(* IEC 61131-3 sources: TwinCATProj/TwinCATRD/PPS_Archive_fb/Cyl, 23 files *)

(* ---- PPS_Cyl.typ ---- *)
(********************************************************************
 * COPYRIGHT -- Pro Pack Systems, Inc.
 ********************************************************************
 * Library: PPS_Cyl
 * File: PPS_Cyl.typ
 * Author: PaulZ
 * Created: April 16, 2012
 ********************************************************************
 * Data types of library PPS_Cyl
 ********************************************************************)

TYPE
	dtCylCntrlInterface2 : 	STRUCT
		I : dtCylCntrl_Inputs2;
		IQ : dtCylCntrl_InOut2;
		Q : dtCylCntrl_Outputs2;
		stSensorExt : dtDebounceInterface;
		stSensorRet : dtDebounceInterface;
	END_STRUCT;
	dtCylCntrlInterface3 : 	STRUCT
		I : dtCylCntrl_Inputs3;
		IQ : dtCylCntrl_InOut3;
		Q : dtCylCntrl_Outputs3;
		stSensorExt : dtDebounceInterface;
		stSensorRet : dtDebounceInterface;
		stErrData : dtCylCntrl_ErrorData;
	END_STRUCT;
	dtCylCntrl_Inputs2 : 	STRUCT
		xEnableFB : BOOL;
		diType : Enum_CylinderType;
		xValveOffRetract : BOOL;
		xAirOk : BOOL;
		xEnManCntrl : BOOL;
		xManCmdA : BOOL;
		xManCmdB : BOOL;
		xManBrake : BOOL;
		xEmergency : BOOL;
		tTravelDel : TIME;
		xFaultReset : BOOL;
	END_STRUCT;
	dtCylCntrl_Inputs3 : 	STRUCT
		xEnableFB : BOOL;
		diType : Enum_CylinderType;
		xValveOffRetract : BOOL;
		xAirOk : BOOL;
		xEnManCntrl : BOOL;
		xManCmdA : BOOL;
		xManCmdB : BOOL;
		xManBrake : BOOL;
		xEmergency : BOOL;
		tTravelDel : TIME;
		sCylName : STRING[80];
	END_STRUCT;
	dtCylCntrl_InOut2 : 	STRUCT
		xExtCmd : BOOL;
		xRetCmd : BOOL;
		xBrakeEn : BOOL;
		xBrakeDis : BOOL;
	END_STRUCT;
	dtCylCntrl_InOut3 : 	STRUCT
		xExtCmd : BOOL;
		xRetCmd : BOOL;
		xBrakeEn : BOOL;
		xBrakeDis : BOOL;
		xFaultReset : BOOL;
	END_STRUCT;
	dtCylCntrl_Outputs2 : 	STRUCT
		xFBActive : BOOL;
		xSVACmd : BOOL;
		xSVBCmd : BOOL;
		xSVBrakeCmd : BOOL;
		xExtended : BOOL;
		xRetracted : BOOL;
		xFaultNoExt : BOOL;
		xFaultNoRet : BOOL;
		tTimeToExtend : TIME;
		tTimeToRetract : TIME;
	END_STRUCT;
	dtCylCntrl_Outputs3 : 	STRUCT
		xFBActive : BOOL;
		xSVACmd : BOOL;
		xSVBCmd : BOOL;
		xSVBrakeCmd : BOOL;
		xExtended : BOOL;
		xRetracted : BOOL;
		xFault : BOOL;
		sFaultText : STRING[80];
		tTimeToExtend : TIME;
		tTimeToRetract : TIME;
	END_STRUCT;
	dtCylCntrl_ErrorData : 	STRUCT
		uiErrorID : UINT;
	END_STRUCT;
	Enum_CylinderType :
		(
		EN_Cyl_1xSV_Basic := 0,
		EN_Cyl_1xSV_Sensored,
		EN_Cyl_2xSV_Basic_NoBrake,
		EN_Cyl_2xSV_Basic_WBrake,
		EN_Cyl_2xSV_Sensored_NoBrake,
		EN_Cyl_2xSV_Sensored_WBrake
		);
END_TYPE

(* ---- FC_CylFM_1xSV_Basic.st ---- *)
(********************************************************************
 * COPYRIGHT -- Pro Pack Systems, Inc.
 ********************************************************************
 * Library: PPS_Cyl
 * File: FC_CylFM_1xSV_Basic.st
 * Author: PaulZ
 * Created: April 18, 2012
 ********************************************************************
 * Implementation of library PPS_Cyl
 ********************************************************************)

(* Monitors Cylinder Fault for Single SV Cylinder *)
FUNCTION FC_CylFM_1xSV_Basic

IF iq_Cyl.I.diType = EN_Cyl_1xSV_Basic THEN

	IF iq_Cyl.Q.xSVACmd THEN
		IF iq_Timer.Q THEN
			IF iq_Cyl.I.xValveOffRetract THEN
				iq_Cyl.Q.xExtended	:= TRUE;
			ELSE
				iq_Cyl.Q.xRetracted	:= TRUE;
			END_IF
			iq_Timer.IN					:= FALSE;
		END_IF
	ELSE
		IF iq_Timer.Q THEN
			IF iq_Cyl.I.xValveOffRetract THEN
				iq_Cyl.Q.xRetracted	:= TRUE;
			ELSE
				iq_Cyl.Q.xExtended	:= TRUE;
				END_IF
			iq_Timer.IN					:= FALSE;
		END_IF
	END_IF

END_IF

END_FUNCTION

(* ---- FC_CylFM_1xSV_Basic3.st ---- *)
(********************************************************************
 * COPYRIGHT -- Pro Pack Systems, Inc.
 ********************************************************************
 * Library: PPS_Cyl
 * File: FC_CylFM_1xSV_Basic.st
 * Author: PaulZ
 * Created: April 18, 2012
 ********************************************************************
 * Implementation of library PPS_Cyl
 ********************************************************************)

(* Monitors Cylinder Fault for Single SV Cylinder *)
FUNCTION FC_CylFM_1xSV_Basic3

IF iq_Cyl.I.diType = EN_Cyl_1xSV_Basic THEN

	IF iq_Cyl.Q.xSVACmd THEN
		IF iq_Timer.Q THEN
			IF iq_Cyl.I.xValveOffRetract THEN
				iq_Cyl.Q.xExtended	:= TRUE;
			ELSE
				iq_Cyl.Q.xRetracted	:= TRUE;
			END_IF
			iq_Timer.IN					:= FALSE;
		END_IF
	ELSE
		IF iq_Timer.Q THEN
			IF iq_Cyl.I.xValveOffRetract THEN
				iq_Cyl.Q.xRetracted	:= TRUE;
			ELSE
				iq_Cyl.Q.xExtended	:= TRUE;
				END_IF
			iq_Timer.IN					:= FALSE;
		END_IF
	END_IF

END_IF

END_FUNCTION

(* ---- FC_CylFM_1xSV_Sensored.st ---- *)
(********************************************************************
 * COPYRIGHT -- Pro Pack Systems, Inc.
 ********************************************************************
 * Library: PPS_Cyl
 * File: FC_CylFM_1xSV_Sensored.st
 * Author: PaulZ
 * Created: April 18, 2012
 ********************************************************************
 * Implementation of library PPS_Cyl
 ********************************************************************)

(* Monitors Cylinder Fault for Single SV Cylinder with Sensors *)
FUNCTION FC_CylFM_1xSV_Sensored

IF iq_Cyl.I.diType = EN_Cyl_1xSV_Sensored THEN

	xFaultSum	:= iq_Cyl.Q.xFaultNoExt OR iq_Cyl.Q.xFaultNoRet;

	IF NOT xFaultSum THEN
		IF iq_Cyl.I.xValveOffRetract THEN
			IF iq_Cyl.Q.xSVACmd THEN
				IF iq_Cyl.stSensorExt.Q.xCmd THEN
					iq_Cyl.Q.xExtended		:= TRUE;
					iq_Cyl.Q.xFaultNoExt		:= FALSE;
					iq_Timer.IN					:= FALSE;
				ELSE
					IF iq_Timer.Q THEN
						iq_Cyl.Q.xExtended	:= FALSE;
						iq_Cyl.Q.xFaultNoExt	:= TRUE;
						iq_Timer.IN				:= FALSE;
					END_IF
				END_IF
			ELSE
				IF iq_Cyl.stSensorRet.Q.xCmd THEN
					iq_Cyl.Q.xRetracted 		:= TRUE;
					iq_Cyl.Q.xFaultNoRet		:= FALSE;
					iq_Timer.IN					:= FALSE;
				ELSE
					IF iq_Timer.Q THEN
						iq_Cyl.Q.xRetracted	:= FALSE;
						iq_Cyl.Q.xFaultNoRet	:= TRUE;
						iq_Timer.IN				:= FALSE;
					END_IF
				END_IF
			END_IF
		ELSE
			IF NOT iq_Cyl.Q.xSVACmd THEN
				IF iq_Cyl.stSensorExt.Q.xCmd THEN
					iq_Cyl.Q.xExtended		:= TRUE;
					iq_Cyl.Q.xFaultNoExt		:= FALSE;
					iq_Timer.IN					:= FALSE;
				ELSE
					IF iq_Timer.Q THEN
						iq_Cyl.Q.xExtended	:= FALSE;
						iq_Cyl.Q.xFaultNoExt	:= TRUE;
						iq_Timer.IN				:= FALSE;
					END_IF
				END_IF
			ELSE
				IF iq_Cyl.stSensorRet.Q.xCmd THEN
					iq_Cyl.Q.xRetracted		:= TRUE;
					iq_Cyl.Q.xFaultNoRet		:= FALSE;
					iq_Timer.IN					:= FALSE;
				ELSE
					IF iq_Timer.Q THEN
						iq_Cyl.Q.xRetracted	:= FALSE;
						iq_Cyl.Q.xFaultNoRet	:= TRUE;
						iq_Timer.IN				:= FALSE;
					END_IF
				END_IF
			END_IF
		END_IF
	END_IF

END_IF

END_FUNCTION

(* ---- FC_CylFM_1xSV_Sensored3.st ---- *)
(********************************************************************
 * COPYRIGHT -- Pro Pack Systems, Inc.
 ********************************************************************
 * Library: PPS_Cyl
 * File: FC_CylFM_1xSV_Sensored.st
 * Author: PaulZ
 * Created: April 18, 2012
 ********************************************************************
 * Implementation of library PPS_Cyl
 ********************************************************************)

(* Monitors Cylinder Fault for Single SV Cylinder with Sensors *)
FUNCTION FC_CylFM_1xSV_Sensored3

IF iq_Cyl.I.diType = EN_Cyl_1xSV_Sensored THEN

	xFaultSum	:= iq_Cyl.Q.xFault;

	IF NOT xFaultSum THEN
		IF iq_Cyl.I.xValveOffRetract THEN
			IF iq_Cyl.Q.xSVACmd THEN
				IF iq_Cyl.stSensorExt.Q.xCmd THEN
					iq_Cyl.Q.xExtended		:= TRUE;
					iq_Cyl.Q.xFault				:= FALSE;
					iq_Cyl.Q.sFaultText		:= '';
					iq_Timer.IN					:= FALSE;
				ELSE
					IF iq_Timer.Q THEN
						iq_Cyl.Q.xExtended			:= FALSE;
						iq_Cyl.Q.xFault					:= TRUE;
						iq_Cyl.Q.sFaultText			:= CONCAT(iq_Cyl.I.sCylName, sNoExtTxt);
						iq_Timer.IN						:= FALSE;
					END_IF
				END_IF
			ELSE
				IF iq_Cyl.stSensorRet.Q.xCmd THEN
					iq_Cyl.Q.xRetracted 		:= TRUE;
					iq_Cyl.Q.xFault				:= FALSE;
					iq_Cyl.Q.sFaultText		:= '';
					iq_Timer.IN					:= FALSE;
				ELSE
					IF iq_Timer.Q THEN
						iq_Cyl.Q.xRetracted			:= FALSE;
						iq_Cyl.Q.xFault					:= TRUE;
						iq_Cyl.Q.sFaultText			:= CONCAT(iq_Cyl.I.sCylName, sNoRetTxt);
						iq_Timer.IN						:= FALSE;
					END_IF
				END_IF
			END_IF
		ELSE
			IF NOT iq_Cyl.Q.xSVACmd THEN
				IF iq_Cyl.stSensorExt.Q.xCmd THEN
					iq_Cyl.Q.xExtended		:= TRUE;
					iq_Cyl.Q.xFault				:= FALSE;
					iq_Cyl.Q.sFaultText		:= '';
					iq_Timer.IN					:= FALSE;
				ELSE
					IF iq_Timer.Q THEN
						iq_Cyl.Q.xExtended			:= FALSE;
						iq_Cyl.Q.xFault					:= TRUE;
						iq_Cyl.Q.sFaultText			:= CONCAT(iq_Cyl.I.sCylName, sNoExtTxt);
						iq_Timer.IN						:= FALSE;
					END_IF
				END_IF
			ELSE
				IF iq_Cyl.stSensorRet.Q.xCmd THEN
					iq_Cyl.Q.xRetracted		:= TRUE;
					iq_Cyl.Q.xFault				:= FALSE;
					iq_Cyl.Q.sFaultText		:= '';
					iq_Timer.IN					:= FALSE;
				ELSE
					IF iq_Timer.Q THEN
						iq_Cyl.Q.xRetracted			:= FALSE;
						iq_Cyl.Q.xFault					:= TRUE;
						iq_Cyl.Q.sFaultText			:= CONCAT(iq_Cyl.I.sCylName, sNoRetTxt);
						iq_Timer.IN						:= FALSE;
					END_IF
				END_IF
			END_IF
		END_IF
	END_IF

END_IF

END_FUNCTION

(* ---- FC_CylFM_2xSV_Basic_NoBrake.st ---- *)
(********************************************************************
 * COPYRIGHT -- Pro Pack Systems, Inc.
 ********************************************************************
 * Library: PPS_Cyl
 * File: FC_CylFM_2xSV_Basic_NoBrake.st
 * Author: PaulZ
 * Created: April 18, 2012
 ********************************************************************
 * Implementation of library PPS_Cyl
 ********************************************************************)

(* Monitors Cylinder Fault for Double SV Cylinder *)
FUNCTION FC_CylFM_2xSV_Basic_NoBrake

IF iq_Cyl.I.diType = EN_Cyl_2xSV_Basic_NoBrake THEN

	IF iq_Cyl.Q.xSVACmd THEN
		IF iq_Timer.Q THEN
			IF iq_Cyl.I.xValveOffRetract THEN
				iq_Cyl.Q.xExtended		:= TRUE;
				iq_Cyl.Q.tTimeToExtend	:= iq_Timer.ET;
			ELSE
				iq_Cyl.Q.xRetracted		:= TRUE;
				iq_Cyl.Q.tTimeToRetract	:= iq_Timer.ET;
			END_IF
			iq_Timer.IN						:= FALSE;
		END_IF
	ELSIF iq_Cyl.Q.xSVBCmd THEN
		IF iq_Timer.Q THEN
			IF iq_Cyl.I.xValveOffRetract THEN
				iq_Cyl.Q.xRetracted		:= TRUE;
				iq_Cyl.Q.tTimeToRetract	:= iq_Timer.ET;
			ELSE
				iq_Cyl.Q.xExtended		:= TRUE;
				iq_Cyl.Q.tTimeToExtend	:= iq_Timer.ET;
 			END_IF
			iq_Timer.IN						:= FALSE;
		END_IF
	END_IF

END_IF

END_FUNCTION

(* ---- FC_CylFM_2xSV_Basic_NoBrake3.st ---- *)
(********************************************************************
 * COPYRIGHT -- Pro Pack Systems, Inc.
 ********************************************************************
 * Library: PPS_Cyl
 * File: FC_CylFM_2xSV_Basic_NoBrake.st
 * Author: PaulZ
 * Created: April 18, 2012
 ********************************************************************
 * Implementation of library PPS_Cyl
 ********************************************************************)

(* Monitors Cylinder Fault for Double SV Cylinder *)
FUNCTION FC_CylFM_2xSV_Basic_NoBrake3

IF iq_Cyl.I.diType = EN_Cyl_2xSV_Basic_NoBrake THEN

	IF iq_Cyl.Q.xSVACmd THEN
		IF iq_Timer.Q THEN
			IF iq_Cyl.I.xValveOffRetract THEN
				iq_Cyl.Q.xExtended		:= TRUE;
				iq_Cyl.Q.tTimeToExtend	:= iq_Timer.ET;
			ELSE
				iq_Cyl.Q.xRetracted		:= TRUE;
				iq_Cyl.Q.tTimeToRetract	:= iq_Timer.ET;
			END_IF
			iq_Timer.IN						:= FALSE;
		END_IF
	ELSIF iq_Cyl.Q.xSVBCmd THEN
		IF iq_Timer.Q THEN
			IF iq_Cyl.I.xValveOffRetract THEN
				iq_Cyl.Q.xRetracted		:= TRUE;
				iq_Cyl.Q.tTimeToRetract	:= iq_Timer.ET;
			ELSE
				iq_Cyl.Q.xExtended		:= TRUE;
				iq_Cyl.Q.tTimeToExtend	:= iq_Timer.ET;
 			END_IF
			iq_Timer.IN						:= FALSE;
		END_IF
	END_IF

END_IF

END_FUNCTION

(* ---- FC_CylFM_2xSV_Basic_wBrake.st ---- *)
(********************************************************************
 * COPYRIGHT -- Pro Pack Systems, Inc.
 ********************************************************************
 * Library: PPS_Cyl
 * File: FC_CylFM_2xSV_Basic_wBrake.st
 * Author: PaulZ
 * Created: April 23, 2012
 ********************************************************************
 * Implementation of library PPS_Cyl
 ********************************************************************)

(* Monitors Cylinder Faults for Double SV Cylinder, no Sensors, with Brake *)
FUNCTION FC_CylFM_2xSV_Basic_wBrake

IF iq_Cyl.I.diType = EN_Cyl_2xSV_Basic_WBrake THEN

	IF iq_Cyl.Q.xSVACmd THEN
		IF iq_Timer.Q THEN
			IF iq_Cyl.I.xValveOffRetract THEN
				iq_Cyl.Q.xExtended		:= TRUE;
				iq_Cyl.Q.tTimeToExtend	:= iq_Timer.ET;
			ELSE
				iq_Cyl.Q.xRetracted		:= TRUE;
				iq_Cyl.Q.tTimeToRetract	:= iq_Timer.ET;
			END_IF
			iq_Timer.IN						:= FALSE;
		END_IF
	ELSIF iq_Cyl.Q.xSVBCmd THEN
		IF iq_Timer.Q THEN
			IF iq_Cyl.I.xValveOffRetract THEN
				iq_Cyl.Q.xRetracted		:= TRUE;
				iq_Cyl.Q.tTimeToRetract	:= iq_Timer.ET;
			ELSE
				iq_Cyl.Q.xExtended		:= TRUE;
				iq_Cyl.Q.tTimeToExtend	:= iq_Timer.ET;
 			END_IF
			iq_Timer.IN						:= FALSE;
		END_IF
	END_IF

END_IF

END_FUNCTION

(* ---- FC_CylFM_2xSV_Basic_wBrake3.st ---- *)
(********************************************************************
 * COPYRIGHT -- Pro Pack Systems, Inc.
 ********************************************************************
 * Library: PPS_Cyl
 * File: FC_CylFM_2xSV_Basic_wBrake.st
 * Author: PaulZ
 * Created: April 23, 2012
 ********************************************************************
 * Implementation of library PPS_Cyl
 ********************************************************************)

(* Monitors Cylinder Faults for Double SV Cylinder, no Sensors, with Brake *)
FUNCTION FC_CylFM_2xSV_Basic_wBrake3

IF iq_Cyl.I.diType = EN_Cyl_2xSV_Basic_WBrake THEN

	IF iq_Cyl.Q.xSVACmd THEN
		IF iq_Timer.Q THEN
			IF iq_Cyl.I.xValveOffRetract THEN
				iq_Cyl.Q.xExtended		:= TRUE;
				iq_Cyl.Q.tTimeToExtend	:= iq_Timer.ET;
			ELSE
				iq_Cyl.Q.xRetracted		:= TRUE;
				iq_Cyl.Q.tTimeToRetract	:= iq_Timer.ET;
			END_IF
			iq_Timer.IN						:= FALSE;
		END_IF
	ELSIF iq_Cyl.Q.xSVBCmd THEN
		IF iq_Timer.Q THEN
			IF iq_Cyl.I.xValveOffRetract THEN
				iq_Cyl.Q.xRetracted		:= TRUE;
				iq_Cyl.Q.tTimeToRetract	:= iq_Timer.ET;
			ELSE
				iq_Cyl.Q.xExtended		:= TRUE;
				iq_Cyl.Q.tTimeToExtend	:= iq_Timer.ET;
 			END_IF
			iq_Timer.IN						:= FALSE;
		END_IF
	END_IF

END_IF

END_FUNCTION

(* ---- FC_CylFM_2xSV_Sensored_NoBrake.st ---- *)
(********************************************************************
 * COPYRIGHT -- Pro Pack Systems, Inc.
 ********************************************************************
 * Library: PPS_Cyl
 * File: FC_CylFM_2xSV_Sensored_NoBrake.st
 * Author: PaulZ
 * Created: April 18, 2012
 ********************************************************************
 * Implementation of library PPS_Cyl
 ********************************************************************)

(* Monitors Cylinder Fault for Double SV Cylinder with Sensor and no Brake *)
FUNCTION FC_CylFM_2xSV_Sensored_NoBrake

IF iq_Cyl.I.diType = EN_Cyl_2xSV_Sensored_NoBrake THEN

	xFaultSum	:= iq_Cyl.Q.xFaultNoExt OR iq_Cyl.Q.xFaultNoRet;

 	IF NOT xFaultSum THEN
		IF iq_Cyl.I.xValveOffRetract THEN
			IF iq_Cyl.Q.xSVACmd THEN
				IF iq_Cyl.stSensorExt.Q.xCmd THEN
					iq_Cyl.Q.xExtended			:= TRUE;
					iq_Cyl.Q.xFaultNoExt			:= FALSE;
					iq_Timer.IN						:= FALSE;
				ELSE
					IF iq_Timer.Q THEN
						iq_Cyl.Q.xExtended		:= FALSE;
						iq_Cyl.Q.xFaultNoExt		:= TRUE;
						iq_Timer.IN					:= FALSE;
					END_IF
				END_IF
			ELSIF iq_Cyl.Q.xSVBCmd THEN
				IF iq_Cyl.stSensorRet.Q.xCmd THEN
					iq_Cyl.Q.xRetracted 			:= TRUE;
					iq_Cyl.Q.xFaultNoRet			:= FALSE;
					iq_Timer.IN						:= FALSE;
				ELSE
					IF iq_Timer.Q THEN
						iq_Cyl.Q.xRetracted		:= FALSE;
						iq_Cyl.Q.xFaultNoRet		:= TRUE;
						iq_Timer.IN					:= FALSE;
					END_IF
				END_IF
			END_IF
		ELSE
			IF iq_Cyl.Q.xSVBCmd THEN
				IF iq_Cyl.stSensorExt.Q.xCmd THEN
					iq_Cyl.Q.xExtended			:= TRUE;
					iq_Cyl.Q.xFaultNoExt			:= FALSE;
					iq_Timer.IN						:= FALSE;
				ELSE
					IF iq_Timer.Q THEN
						iq_Cyl.Q.xExtended		:= FALSE;
						iq_Cyl.Q.xFaultNoExt		:= TRUE;
						iq_Timer.IN					:= FALSE;
					END_IF
				END_IF
			ELSIF iq_Cyl.Q.xSVACmd THEN
				IF iq_Cyl.stSensorRet.Q.xCmd THEN
					iq_Cyl.Q.xRetracted			:= TRUE;
					iq_Cyl.Q.xFaultNoRet			:= FALSE;
					iq_Timer.IN						:= FALSE;
				ELSE
					IF iq_Timer.Q THEN
						iq_Cyl.Q.xRetracted		:= FALSE;
						iq_Cyl.Q.xFaultNoRet		:= TRUE;
						iq_Timer.IN					:= FALSE;
					END_IF
				END_IF
			END_IF
		END_IF
	END_IF

END_IF

END_FUNCTION

(* ---- FC_CylFM_2xSV_Sensored_NoBrake3.st ---- *)
(********************************************************************
 * COPYRIGHT -- Pro Pack Systems, Inc.
 ********************************************************************
 * Library: PPS_Cyl
 * File: FC_CylFM_2xSV_Sensored_NoBrake.st
 * Author: PaulZ
 * Created: April 18, 2012
 ********************************************************************
 * Implementation of library PPS_Cyl
 ********************************************************************)

(* Monitors Cylinder Fault for Double SV Cylinder with Sensor and no Brake *)
FUNCTION FC_CylFM_2xSV_Sensored_NoBrake3

IF iq_Cyl.I.diType = EN_Cyl_2xSV_Sensored_NoBrake THEN

	xFaultSum	:= iq_Cyl.Q.xFault;

 	IF NOT xFaultSum THEN
		IF iq_Cyl.I.xValveOffRetract THEN
			IF iq_Cyl.Q.xSVACmd THEN
				IF iq_Cyl.stSensorExt.Q.xCmd THEN
					iq_Cyl.Q.xExtended			:= TRUE;
					iq_Cyl.Q.xFault					:= FALSE;
					iq_Cyl.Q.sFaultText			:= '';
					iq_Timer.IN						:= FALSE;
				ELSE
					IF iq_Timer.Q THEN
						iq_Cyl.Q.xExtended			:= FALSE;
						iq_Cyl.Q.xFault					:= TRUE;
						iq_Cyl.Q.sFaultText			:= CONCAT(iq_Cyl.I.sCylName, sNoExtTxt);
						iq_Timer.IN						:= FALSE;
					END_IF
				END_IF
			ELSIF iq_Cyl.Q.xSVBCmd THEN
				IF iq_Cyl.stSensorRet.Q.xCmd THEN
					iq_Cyl.Q.xRetracted 			:= TRUE;
					iq_Cyl.Q.xFault					:= FALSE;
					iq_Cyl.Q.sFaultText			:= '';
					iq_Timer.IN						:= FALSE;
				ELSE
					IF iq_Timer.Q THEN
						iq_Cyl.Q.xRetracted			:= FALSE;
						iq_Cyl.Q.xFault					:= TRUE;
						iq_Cyl.Q.sFaultText			:= CONCAT(iq_Cyl.I.sCylName, sNoRetTxt);
						iq_Timer.IN						:= FALSE;
					END_IF
				END_IF
			END_IF
		ELSE
			IF iq_Cyl.Q.xSVBCmd THEN
				IF iq_Cyl.stSensorExt.Q.xCmd THEN
					iq_Cyl.Q.xExtended			:= TRUE;
					iq_Cyl.Q.xFault					:= FALSE;
					iq_Cyl.Q.sFaultText			:= '';
					iq_Timer.IN						:= FALSE;
				ELSE
					IF iq_Timer.Q THEN
						iq_Cyl.Q.xExtended			:= FALSE;
						iq_Cyl.Q.xFault					:= TRUE;
						iq_Cyl.Q.sFaultText			:= CONCAT(iq_Cyl.I.sCylName, sNoExtTxt);
						iq_Timer.IN						:= FALSE;
					END_IF
				END_IF
			ELSIF iq_Cyl.Q.xSVACmd THEN
				IF iq_Cyl.stSensorRet.Q.xCmd THEN
					iq_Cyl.Q.xRetracted			:= TRUE;
					iq_Cyl.Q.xFault					:= FALSE;
					iq_Cyl.Q.sFaultText			:= '';
					iq_Timer.IN						:= FALSE;
				ELSE
					IF iq_Timer.Q THEN
						iq_Cyl.Q.xRetracted			:= FALSE;
						iq_Cyl.Q.xFault					:= TRUE;
						iq_Cyl.Q.sFaultText			:= CONCAT(iq_Cyl.I.sCylName, sNoRetTxt);
						iq_Timer.IN						:= FALSE;
					END_IF
				END_IF
			END_IF
		END_IF
	END_IF

END_IF

END_FUNCTION

(* ---- FC_CylFM_2xSV_Sensored_wBrake.st ---- *)
(********************************************************************
 * COPYRIGHT -- Pro Pack Systems, Inc.
 ********************************************************************
 * Library: PPS_Cyl
 * File: FC_CylFM_2xSV_Sensored_wBrake.st
 * Author: PaulZ
 * Created: April 18, 2012
 ********************************************************************
 * Implementation of library PPS_Cyl
 ********************************************************************)

(* Monitors Cylinder Fault for Double SV Cylinder with Sensors and Brake *)
FUNCTION FC_CylFM_2xSV_Sensored_wBrake

IF iq_Cyl.I.diType = EN_Cyl_2xSV_Sensored_WBrake THEN

	xFaultSum	:= iq_Cyl.Q.xFaultNoExt OR iq_Cyl.Q.xFaultNoRet;

 	IF iq_Cyl.Q.xSVBrakeCmd THEN
 		iq_Timer.IN		:= FALSE;
	END_IF

	IF NOT xFaultSum THEN
		IF iq_Cyl.I.xValveOffRetract THEN
			IF iq_Cyl.Q.xSVACmd THEN
				IF iq_Cyl.stSensorExt.Q.xCmd THEN
					iq_Cyl.Q.xExtended			:= TRUE;
					iq_Cyl.Q.xFaultNoExt			:= FALSE;
					iq_Timer.IN						:= FALSE;
				ELSE
					IF iq_Timer.Q THEN
						iq_Cyl.Q.xExtended		:= FALSE;
						iq_Cyl.Q.xFaultNoExt		:= TRUE;
						iq_Timer.IN					:= FALSE;
					END_IF
				END_IF
			ELSIF iq_Cyl.Q.xSVBCmd THEN
				IF iq_Cyl.stSensorRet.Q.xCmd THEN
					iq_Cyl.Q.xRetracted 			:= TRUE;
					iq_Cyl.Q.xFaultNoRet			:= FALSE;
					iq_Timer.IN						:= FALSE;
				ELSE
					IF iq_Timer.Q THEN
						iq_Cyl.Q.xRetracted		:= FALSE;
						iq_Cyl.Q.xFaultNoRet		:= TRUE;
						iq_Timer.IN					:= FALSE;
					END_IF
				END_IF
			END_IF
		ELSE
			IF iq_Cyl.Q.xSVBCmd THEN
				IF iq_Cyl.stSensorExt.Q.xCmd THEN
					iq_Cyl.Q.xExtended			:= TRUE;
					iq_Cyl.Q.xFaultNoExt			:= FALSE;
					iq_Timer.IN						:= FALSE;
				ELSE
					IF iq_Timer.Q THEN
						iq_Cyl.Q.xExtended		:= FALSE;
						iq_Cyl.Q.xFaultNoExt		:= TRUE;
						iq_Timer.IN					:= FALSE;
					END_IF
				END_IF
			ELSIF iq_Cyl.Q.xSVACmd THEN
				IF iq_Cyl.stSensorRet.Q.xCmd THEN
					iq_Cyl.Q.xRetracted			:= TRUE;
					iq_Cyl.Q.xFaultNoRet			:= FALSE;
					iq_Timer.IN						:= FALSE;
				ELSE
					IF iq_Timer.Q THEN
						iq_Cyl.Q.xRetracted		:= FALSE;
						iq_Cyl.Q.xFaultNoRet		:= TRUE;
						iq_Timer.IN					:= FALSE;
					END_IF
				END_IF
			END_IF
		END_IF
	END_IF

END_IF

END_FUNCTION

(* ---- FC_CylFM_2xSV_Sensored_wBrake3.st ---- *)
(********************************************************************
 * COPYRIGHT -- Pro Pack Systems, Inc.
 ********************************************************************
 * Library: PPS_Cyl
 * File: FC_CylFM_2xSV_Sensored_wBrake.st
 * Author: PaulZ
 * Created: April 18, 2012
 ********************************************************************
 * Implementation of library PPS_Cyl
 ********************************************************************)

(* Monitors Cylinder Fault for Double SV Cylinder with Sensors and Brake *)
FUNCTION FC_CylFM_2xSV_Sensored_wBrake3

IF iq_Cyl.I.diType = EN_Cyl_2xSV_Sensored_WBrake THEN

	xFaultSum	:= iq_Cyl.Q.xFault;

 	IF iq_Cyl.Q.xSVBrakeCmd THEN
 		iq_Timer.IN		:= FALSE;
	END_IF

	IF NOT xFaultSum THEN
		IF iq_Cyl.I.xValveOffRetract THEN
			IF iq_Cyl.Q.xSVACmd THEN
				IF iq_Cyl.stSensorExt.Q.xCmd THEN
					iq_Cyl.Q.xExtended			:= TRUE;
					iq_Cyl.Q.xFault					:= FALSE;
					iq_Cyl.Q.sFaultText			:= '';
					iq_Timer.IN						:= FALSE;
				ELSE
					IF iq_Timer.Q THEN
						iq_Cyl.Q.xExtended			:= FALSE;
						iq_Cyl.Q.xFault					:= TRUE;
						iq_Cyl.Q.sFaultText			:= CONCAT(iq_Cyl.I.sCylName, sNoExtTxt);
						iq_Timer.IN						:= FALSE;
					END_IF
				END_IF
			ELSIF iq_Cyl.Q.xSVBCmd THEN
				IF iq_Cyl.stSensorRet.Q.xCmd THEN
					iq_Cyl.Q.xRetracted 			:= TRUE;
					iq_Cyl.Q.xFault					:= FALSE;
					iq_Cyl.Q.sFaultText			:= '';
					iq_Timer.IN						:= FALSE;
				ELSE
					IF iq_Timer.Q THEN
						iq_Cyl.Q.xRetracted			:= FALSE;
						iq_Cyl.Q.xFault					:= TRUE;
						iq_Cyl.Q.sFaultText			:= CONCAT(iq_Cyl.I.sCylName, sNoRetTxt);
						iq_Timer.IN						:= FALSE;
					END_IF
				END_IF
			END_IF
		ELSE
			IF iq_Cyl.Q.xSVBCmd THEN
				IF iq_Cyl.stSensorExt.Q.xCmd THEN
					iq_Cyl.Q.xExtended			:= TRUE;
					iq_Cyl.Q.xFault					:= FALSE;
					iq_Cyl.Q.sFaultText			:= '';
					iq_Timer.IN						:= FALSE;
				ELSE
					IF iq_Timer.Q THEN
						iq_Cyl.Q.xExtended			:= FALSE;
						iq_Cyl.Q.xFault					:= TRUE;
						iq_Cyl.Q.sFaultText			:= CONCAT(iq_Cyl.I.sCylName, sNoExtTxt);
						iq_Timer.IN						:= FALSE;
					END_IF
				END_IF
			ELSIF iq_Cyl.Q.xSVACmd THEN
				IF iq_Cyl.stSensorRet.Q.xCmd THEN
					iq_Cyl.Q.xRetracted			:= TRUE;
					iq_Cyl.Q.xFault					:= FALSE;
					iq_Cyl.Q.sFaultText			:= '';
					iq_Timer.IN						:= FALSE;
				ELSE
					IF iq_Timer.Q THEN
						iq_Cyl.Q.xRetracted			:= FALSE;
						iq_Cyl.Q.xFault					:= TRUE;
						iq_Cyl.Q.sFaultText			:= CONCAT(iq_Cyl.I.sCylName, sNoRetTxt);
						iq_Timer.IN						:= FALSE;
					END_IF
				END_IF
			END_IF
		END_IF
	END_IF

END_IF

END_FUNCTION

(* ---- FC_CylQ_1xSV.st ---- *)
(********************************************************************
 * COPYRIGHT -- Pro Pack Systems, Inc.
 ********************************************************************
 * Library: PPS_Cyl
 * File: FC_CylQ_1xSV_Basic.st
 * Author: PaulZ
 * Created: April 19, 2012
 ********************************************************************
 * Implementation of library PPS_Cyl
 ********************************************************************)

(* Controls the outputs for a Single SV Cylinder *)
FUNCTION FC_CylQ_1xSV

IF iq_Cyl.I.diType = EN_Cyl_1xSV_Basic OR
	iq_Cyl.I.diType = EN_Cyl_1xSV_Sensored THEN

	IF NOT iq_Cyl.I.xEnManCntrl THEN (* When not in Manual Mode, control output *)

		IF iq_Cyl.I.xValveOffRetract THEN
			IF iq_Cyl.IQ.xExtCmd THEN
				iq_Cyl.Q.xSVACmd		:= TRUE;
				iq_Cyl.Q.xRetracted		:= FALSE;
				iq_Cyl.Q.xExtended		:= FALSE;
				iq_Cyl.Q.tTimeToExtend	:= T#0ms;
				iq_Timer.IN					:= TRUE;
				IF iq_Cyl.Q.xSVACmd THEN
					iq_Cyl.IQ.xExtCmd		:= FALSE;
				END_IF
			END_IF

			IF iq_Cyl.IQ.xRetCmd THEN
				iq_Cyl.Q.xSVACmd		:= FALSE;
				iq_Cyl.Q.xExtended		:= FALSE;
				iq_Cyl.Q.xRetracted		:= FALSE;
				iq_Cyl.Q.tTimeToRetract	:= T#0ms;
				iq_Timer.IN					:= TRUE;
				IF NOT iq_Cyl.Q.xSVACmd THEN
					iq_Cyl.IQ.xRetCmd		:= FALSE;
				END_IF
			END_IF
		ELSE
			IF iq_Cyl.IQ.xExtCmd THEN
				iq_Cyl.Q.xSVACmd		:= FALSE;
				iq_Cyl.Q.xExtended		:= FALSE;
				iq_Cyl.Q.xRetracted		:= FALSE;
				iq_Cyl.Q.tTimeToExtend	:= T#0ms;
				iq_Timer.IN					:= TRUE;
				IF NOT iq_Cyl.Q.xSVACmd THEN
					iq_Cyl.IQ.xExtCmd		:= FALSE;
				END_IF
			END_IF

			IF iq_Cyl.IQ.xRetCmd THEN
				iq_Cyl.Q.xSVACmd		:= TRUE;
				iq_Cyl.Q.xExtended		:= FALSE;
				iq_Cyl.Q.xRetracted		:= FALSE;
				iq_Cyl.Q.tTimeToRetract	:= T#0ms;
				iq_Timer.IN					:= TRUE;
				IF iq_Cyl.Q.xSVACmd THEN
					iq_Cyl.IQ.xRetCmd		:= FALSE;
				END_IF
			END_IF
		END_IF

	ELSE (* When in Manual Mode, control output *)
		IF iq_Cyl.Q.xSVACmd THEN
			IF xManCmd THEN
				iq_Cyl.Q.xSVACmd		:= FALSE;
				iq_Cyl.Q.xRetracted		:= FALSE;
				iq_Cyl.Q.xExtended		:= FALSE;
				iq_Cyl.Q.tTimeToRetract	:= T#0ms;
				iq_Timer.IN					:= TRUE;
			END_IF
		ELSE
			IF xManCmd THEN
				iq_Cyl.Q.xSVACmd		:= TRUE;
				iq_Cyl.Q.xRetracted		:= FALSE;
				iq_Cyl.Q.xExtended		:= FALSE;
				iq_Cyl.Q.tTimeToExtend	:= T#0ms;
				iq_Timer.IN					:= TRUE;
			END_IF
		END_IF
	END_IF

END_IF

END_FUNCTION

(* ---- FC_CylQ_1xSV3.st ---- *)
(********************************************************************
 * COPYRIGHT -- Pro Pack Systems, Inc.
 ********************************************************************
 * Library: PPS_Cyl
 * File: FC_CylQ_1xSV_Basic.st
 * Author: PaulZ
 * Created: April 19, 2012
 ********************************************************************
 * Implementation of library PPS_Cyl
 ********************************************************************)

(* Controls the outputs for a Single SV Cylinder *)
FUNCTION FC_CylQ_1xSV3

IF iq_Cyl.I.diType = EN_Cyl_1xSV_Basic OR
	iq_Cyl.I.diType = EN_Cyl_1xSV_Sensored THEN

	IF NOT iq_Cyl.I.xEnManCntrl THEN (* When not in Manual Mode, control output *)

		IF iq_Cyl.I.xValveOffRetract THEN
			IF iq_Cyl.IQ.xExtCmd THEN
				iq_Cyl.Q.xSVACmd		:= TRUE;
				iq_Cyl.Q.xRetracted		:= FALSE;
				iq_Cyl.Q.xExtended		:= FALSE;
				iq_Cyl.Q.tTimeToExtend	:= T#0ms;
				iq_Timer.IN					:= TRUE;
				IF iq_Cyl.Q.xSVACmd THEN
					iq_Cyl.IQ.xExtCmd		:= FALSE;
				END_IF
			END_IF

			IF iq_Cyl.IQ.xRetCmd THEN
				iq_Cyl.Q.xSVACmd		:= FALSE;
				iq_Cyl.Q.xExtended		:= FALSE;
				iq_Cyl.Q.xRetracted		:= FALSE;
				iq_Cyl.Q.tTimeToRetract	:= T#0ms;
				iq_Timer.IN					:= TRUE;
				IF NOT iq_Cyl.Q.xSVACmd THEN
					iq_Cyl.IQ.xRetCmd		:= FALSE;
				END_IF
			END_IF
		ELSE
			IF iq_Cyl.IQ.xExtCmd THEN
				iq_Cyl.Q.xSVACmd		:= FALSE;
				iq_Cyl.Q.xExtended		:= FALSE;
				iq_Cyl.Q.xRetracted		:= FALSE;
				iq_Cyl.Q.tTimeToExtend	:= T#0ms;
				iq_Timer.IN					:= TRUE;
				IF NOT iq_Cyl.Q.xSVACmd THEN
					iq_Cyl.IQ.xExtCmd		:= FALSE;
				END_IF
			END_IF

			IF iq_Cyl.IQ.xRetCmd THEN
				iq_Cyl.Q.xSVACmd		:= TRUE;
				iq_Cyl.Q.xExtended		:= FALSE;
				iq_Cyl.Q.xRetracted		:= FALSE;
				iq_Cyl.Q.tTimeToRetract	:= T#0ms;
				iq_Timer.IN					:= TRUE;
				IF iq_Cyl.Q.xSVACmd THEN
					iq_Cyl.IQ.xRetCmd		:= FALSE;
				END_IF
			END_IF
		END_IF

	ELSE (* When in Manual Mode, control output *)
		IF iq_Cyl.Q.xSVACmd THEN
			IF xManCmd THEN
				iq_Cyl.Q.xSVACmd		:= FALSE;
				iq_Cyl.Q.xRetracted		:= FALSE;
				iq_Cyl.Q.xExtended		:= FALSE;
				iq_Cyl.Q.tTimeToRetract	:= T#0ms;
				iq_Timer.IN					:= TRUE;
			END_IF
		ELSE
			IF xManCmd THEN
				iq_Cyl.Q.xSVACmd		:= TRUE;
				iq_Cyl.Q.xRetracted		:= FALSE;
				iq_Cyl.Q.xExtended		:= FALSE;
				iq_Cyl.Q.tTimeToExtend	:= T#0ms;
				iq_Timer.IN					:= TRUE;
			END_IF
		END_IF
	END_IF

END_IF

END_FUNCTION

(* ---- FC_CylQ_2xSV_NoBrake.st ---- *)
(********************************************************************
 * COPYRIGHT -- Pro Pack Systems, Inc.
 ********************************************************************
 * Library: PPS_Cyl
 * File: FC_CylQ_1xSV_Basic.st
 * Author: PaulZ
 * Created: April 19, 2012
 ********************************************************************
 * Implementation of library PPS_Cyl
 ********************************************************************)

(* Controls the outputs for a Double SV Cylinder, no Brake *)
FUNCTION FC_CylQ_2xSV_NoBrake

IF iq_Cyl.I.diType = EN_Cyl_2xSV_Basic_NoBrake OR
	iq_Cyl.I.diType = EN_Cyl_2xSV_Sensored_NoBrake THEN

	IF NOT iq_Cyl.I.xEnManCntrl THEN (* When not in Manual Mode, control output *)

		IF iq_Cyl.I.xValveOffRetract THEN
			IF iq_Cyl.IQ.xExtCmd THEN
				iq_Cyl.Q.xSVACmd		:= TRUE;
				iq_Cyl.Q.xSVBCmd		:= FALSE;
				iq_Cyl.Q.xRetracted		:= FALSE;
				iq_Cyl.Q.xExtended		:= FALSE;
				iq_Cyl.Q.tTimeToExtend	:= T#0ms;
				iq_Timer.IN					:= TRUE;
				IF iq_Cyl.Q.xSVACmd AND NOT iq_Cyl.Q.xSVBCmd THEN
					iq_Cyl.IQ.xExtCmd		:= FALSE;
				END_IF
			END_IF

			IF iq_Cyl.IQ.xRetCmd THEN
				iq_Cyl.Q.xSVACmd		:= FALSE;
				iq_Cyl.Q.xSVBCmd		:= TRUE;
				iq_Cyl.Q.xExtended		:= FALSE;
				iq_Cyl.Q.xRetracted		:= FALSE;
				iq_Cyl.Q.tTimeToRetract	:= T#0ms;
				iq_Timer.IN					:= TRUE;
				IF NOT iq_Cyl.Q.xSVACmd AND iq_Cyl.Q.xSVBCmd THEN
					iq_Cyl.IQ.xRetCmd		:= FALSE;
				END_IF
			END_IF
		ELSE
			IF iq_Cyl.IQ.xExtCmd THEN
				iq_Cyl.Q.xSVACmd		:= FALSE;
				iq_Cyl.Q.xSVBCmd		:= TRUE;
				iq_Cyl.Q.xExtended		:= FALSE;
				iq_Cyl.Q.xRetracted		:= FALSE;
				iq_Cyl.Q.tTimeToExtend	:= T#0ms;
				iq_Timer.IN					:= TRUE;
				IF NOT iq_Cyl.Q.xSVACmd AND iq_Cyl.Q.xSVBCmd THEN
					iq_Cyl.IQ.xExtCmd		:= FALSE;
				END_IF
			END_IF

			IF iq_Cyl.IQ.xRetCmd THEN
				iq_Cyl.Q.xSVACmd		:= TRUE;
				iq_Cyl.Q.xSVBCmd		:= FALSE;
				iq_Cyl.Q.xExtended		:= FALSE;
				iq_Cyl.Q.xRetracted		:= FALSE;
				iq_Cyl.Q.tTimeToRetract	:= T#0ms;
				iq_Timer.IN					:= TRUE;
				IF iq_Cyl.Q.xSVACmd AND NOT iq_Cyl.Q.xSVBCmd THEN
					iq_Cyl.IQ.xRetCmd		:= FALSE;
				END_IF
			END_IF
		END_IF

	ELSE (* When in Manual Mode, control output *)
		IF iq_Cyl.Q.xSVACmd THEN
			IF xManCmd THEN
				iq_Cyl.Q.xSVACmd		:= FALSE;
				iq_Cyl.Q.xRetracted		:= FALSE;
				iq_Cyl.Q.xExtended		:= FALSE;
				iq_Timer.IN					:= TRUE;
			END_IF
		ELSE
			IF xManCmd THEN
				iq_Cyl.Q.xSVACmd		:= TRUE;
				iq_Cyl.Q.xSVBCmd		:= FALSE;
				iq_Cyl.Q.xRetracted		:= FALSE;
				iq_Cyl.Q.xExtended		:= FALSE;
				IF iq_Cyl.I.xValveOffRetract THEN
					iq_Cyl.Q.tTimeToExtend	:= T#0ms;
				ELSE
					iq_Cyl.Q.tTimeToRetract	:= T#0ms;
	 			END_IF
				iq_Timer.IN					:= TRUE;
			END_IF
		END_IF

		IF iq_Cyl.Q.xSVBCmd THEN
			IF xManCmdB THEN
				iq_Cyl.Q.xSVBCmd		:= FALSE;
				iq_Cyl.Q.xRetracted		:= FALSE;
				iq_Cyl.Q.xExtended		:= FALSE;
				iq_Timer.IN					:= TRUE;
			END_IF
		ELSE
			IF xManCmdB THEN
				iq_Cyl.Q.xSVBCmd		:= TRUE;
				iq_Cyl.Q.xSVACmd		:= FALSE;
				iq_Cyl.Q.xRetracted		:= FALSE;
				iq_Cyl.Q.xExtended		:= FALSE;
				IF iq_Cyl.I.xValveOffRetract THEN
					iq_Cyl.Q.tTimeToRetract	:= T#0ms;
				ELSE
					iq_Cyl.Q.tTimeToExtend	:= T#0ms;
	 			END_IF
				iq_Timer.IN					:= TRUE;
			END_IF
		END_IF
	END_IF

END_IF

END_FUNCTION

(* ---- FC_CylQ_2xSV_NoBrake3.st ---- *)
(********************************************************************
 * COPYRIGHT -- Pro Pack Systems, Inc.
 ********************************************************************
 * Library: PPS_Cyl
 * File: FC_CylQ_1xSV_Basic.st
 * Author: PaulZ
 * Created: April 19, 2012
 ********************************************************************
 * Implementation of library PPS_Cyl
 ********************************************************************)

(* Controls the outputs for a Double SV Cylinder, no Brake *)
FUNCTION FC_CylQ_2xSV_NoBrake3

IF iq_Cyl.I.diType = EN_Cyl_2xSV_Basic_NoBrake OR
	iq_Cyl.I.diType = EN_Cyl_2xSV_Sensored_NoBrake THEN

	IF NOT iq_Cyl.I.xEnManCntrl THEN (* When not in Manual Mode, control output *)

		IF iq_Cyl.I.xValveOffRetract THEN
			IF iq_Cyl.IQ.xExtCmd THEN
				iq_Cyl.Q.xSVACmd		:= TRUE;
				iq_Cyl.Q.xSVBCmd		:= FALSE;
				iq_Cyl.Q.xRetracted		:= FALSE;
				iq_Cyl.Q.xExtended		:= FALSE;
				iq_Cyl.Q.tTimeToExtend	:= T#0ms;
				iq_Timer.IN					:= TRUE;
				IF iq_Cyl.Q.xSVACmd AND NOT iq_Cyl.Q.xSVBCmd THEN
					iq_Cyl.IQ.xExtCmd		:= FALSE;
				END_IF
			END_IF

			IF iq_Cyl.IQ.xRetCmd THEN
				iq_Cyl.Q.xSVACmd		:= FALSE;
				iq_Cyl.Q.xSVBCmd		:= TRUE;
				iq_Cyl.Q.xExtended		:= FALSE;
				iq_Cyl.Q.xRetracted		:= FALSE;
				iq_Cyl.Q.tTimeToRetract	:= T#0ms;
				iq_Timer.IN					:= TRUE;
				IF NOT iq_Cyl.Q.xSVACmd AND iq_Cyl.Q.xSVBCmd THEN
					iq_Cyl.IQ.xRetCmd		:= FALSE;
				END_IF
			END_IF
		ELSE
			IF iq_Cyl.IQ.xExtCmd THEN
				iq_Cyl.Q.xSVACmd		:= FALSE;
				iq_Cyl.Q.xSVBCmd		:= TRUE;
				iq_Cyl.Q.xExtended		:= FALSE;
				iq_Cyl.Q.xRetracted		:= FALSE;
				iq_Cyl.Q.tTimeToExtend	:= T#0ms;
				iq_Timer.IN					:= TRUE;
				IF NOT iq_Cyl.Q.xSVACmd AND iq_Cyl.Q.xSVBCmd THEN
					iq_Cyl.IQ.xExtCmd		:= FALSE;
				END_IF
			END_IF

			IF iq_Cyl.IQ.xRetCmd THEN
				iq_Cyl.Q.xSVACmd		:= TRUE;
				iq_Cyl.Q.xSVBCmd		:= FALSE;
				iq_Cyl.Q.xExtended		:= FALSE;
				iq_Cyl.Q.xRetracted		:= FALSE;
				iq_Cyl.Q.tTimeToRetract	:= T#0ms;
				iq_Timer.IN					:= TRUE;
				IF iq_Cyl.Q.xSVACmd AND NOT iq_Cyl.Q.xSVBCmd THEN
					iq_Cyl.IQ.xRetCmd		:= FALSE;
				END_IF
			END_IF
		END_IF

	ELSE (* When in Manual Mode, control output *)
		IF iq_Cyl.Q.xSVACmd THEN
			IF xManCmd THEN
				iq_Cyl.Q.xSVACmd		:= FALSE;
				iq_Cyl.Q.xRetracted		:= FALSE;
				iq_Cyl.Q.xExtended		:= FALSE;
				iq_Timer.IN					:= TRUE;
			END_IF
		ELSE
			IF xManCmd THEN
				iq_Cyl.Q.xSVACmd		:= TRUE;
				iq_Cyl.Q.xSVBCmd		:= FALSE;
				iq_Cyl.Q.xRetracted		:= FALSE;
				iq_Cyl.Q.xExtended		:= FALSE;
				IF iq_Cyl.I.xValveOffRetract THEN
					iq_Cyl.Q.tTimeToExtend	:= T#0ms;
				ELSE
					iq_Cyl.Q.tTimeToRetract	:= T#0ms;
	 			END_IF
				iq_Timer.IN					:= TRUE;
			END_IF
		END_IF

		IF iq_Cyl.Q.xSVBCmd THEN
			IF xManCmdB THEN
				iq_Cyl.Q.xSVBCmd		:= FALSE;
				iq_Cyl.Q.xRetracted		:= FALSE;
				iq_Cyl.Q.xExtended		:= FALSE;
				iq_Timer.IN					:= TRUE;
			END_IF
		ELSE
			IF xManCmdB THEN
				iq_Cyl.Q.xSVBCmd		:= TRUE;
				iq_Cyl.Q.xSVACmd		:= FALSE;
				iq_Cyl.Q.xRetracted		:= FALSE;
				iq_Cyl.Q.xExtended		:= FALSE;
				IF iq_Cyl.I.xValveOffRetract THEN
					iq_Cyl.Q.tTimeToRetract	:= T#0ms;
				ELSE
					iq_Cyl.Q.tTimeToExtend	:= T#0ms;
	 			END_IF
				iq_Timer.IN					:= TRUE;
			END_IF
		END_IF
	END_IF

END_IF

END_FUNCTION

(* ---- FC_CylQ_2xSV_wBrake.st ---- *)
(********************************************************************
 * COPYRIGHT -- Pro Pack Systems, Inc.
 ********************************************************************
 * Library: PPS_Cyl
 * File: FC_CylQ_1xSV_Basic.st
 * Author: PaulZ
 * Created: April 19, 2012
 ********************************************************************
 * Implementation of library PPS_Cyl
 ********************************************************************)

(* Controls the outputs for a Double SV Cylinder, with Brake *)
FUNCTION FC_CylQ_2xSV_wBrake

IF iq_Cyl.I.diType = EN_Cyl_2xSV_Basic_WBrake OR
	iq_Cyl.I.diType = EN_Cyl_2xSV_Sensored_WBrake THEN

	IF NOT iq_Cyl.I.xEnManCntrl THEN (* When not in Manual Mode, control output *)

		IF iq_Cyl.IQ.xBrakeEn THEN
  			iq_Cyl.Q.xSVACmd		:= FALSE;
   			iq_Cyl.Q.xSVBCmd		:= FALSE;
   			iq_Cyl.Q.xSVBrakeCmd	:= TRUE;
			iq_Timer.IN					:= FALSE;
			iq_Cyl.IQ.xBrakeEn		:= FALSE;
   		END_IF

		IF iq_Cyl.IQ.xBrakeDis THEN
  			iq_Cyl.Q.xSVBrakeCmd	:= FALSE;
   			iq_Cyl.IQ.xBrakeDis		:= FALSE;
   		END_IF

		IF iq_Cyl.Q.xSVBrakeCmd THEN
  			iq_Cyl.IQ.xExtCmd		:= FALSE;
   			iq_Cyl.IQ.xRetCmd		:= FALSE;
   		END_IF

		IF iq_Cyl.I.xValveOffRetract THEN
			IF iq_Cyl.IQ.xExtCmd THEN
				iq_Cyl.Q.xSVACmd		:= TRUE;
				iq_Cyl.Q.xSVBCmd		:= FALSE;
				iq_Cyl.Q.xRetracted		:= FALSE;
				iq_Cyl.Q.xExtended		:= FALSE;
				iq_Cyl.Q.tTimeToExtend	:= T#0ms;
				iq_Timer.IN					:= TRUE;
				IF iq_Cyl.Q.xSVACmd AND NOT iq_Cyl.Q.xSVBCmd THEN
					iq_Cyl.IQ.xExtCmd		:= FALSE;
				END_IF
			END_IF

			IF iq_Cyl.IQ.xRetCmd THEN
				iq_Cyl.Q.xSVACmd		:= FALSE;
				iq_Cyl.Q.xSVBCmd		:= TRUE;
				iq_Cyl.Q.xExtended		:= FALSE;
				iq_Cyl.Q.xRetracted		:= FALSE;
				iq_Cyl.Q.tTimeToRetract	:= T#0ms;
				iq_Timer.IN					:= TRUE;
				IF NOT iq_Cyl.Q.xSVACmd AND iq_Cyl.Q.xSVBCmd THEN
					iq_Cyl.IQ.xRetCmd		:= FALSE;
				END_IF
			END_IF
		ELSE
			IF iq_Cyl.IQ.xExtCmd THEN
				iq_Cyl.Q.xSVACmd		:= FALSE;
				iq_Cyl.Q.xSVBCmd		:= TRUE;
				iq_Cyl.Q.xExtended		:= FALSE;
				iq_Cyl.Q.xRetracted		:= FALSE;
				iq_Cyl.Q.tTimeToExtend	:= T#0ms;
				iq_Timer.IN					:= TRUE;
				IF NOT iq_Cyl.Q.xSVACmd AND iq_Cyl.Q.xSVBCmd THEN
					iq_Cyl.IQ.xExtCmd		:= FALSE;
				END_IF
			END_IF

			IF iq_Cyl.IQ.xRetCmd THEN
				iq_Cyl.Q.xSVACmd		:= TRUE;
				iq_Cyl.Q.xSVBCmd		:= FALSE;
				iq_Cyl.Q.xExtended		:= FALSE;
				iq_Cyl.Q.xRetracted		:= FALSE;
				iq_Cyl.Q.tTimeToRetract	:= T#0ms;
				iq_Timer.IN					:= TRUE;
				IF iq_Cyl.Q.xSVACmd AND NOT iq_Cyl.Q.xSVBCmd THEN
					iq_Cyl.IQ.xRetCmd		:= FALSE;
				END_IF
			END_IF
		END_IF

	ELSE (* When in Manual Mode, control output *)

		IF xManBrake THEN
  			IF iq_Cyl.Q.xSVBrakeCmd THEN
   				iq_Cyl.Q.xSVBrakeCmd	:= FALSE;
			ELSE
			  	iq_Cyl.Q.xSVBrakeCmd	:= TRUE;
				iq_Cyl.Q.xSVACmd		:= FALSE;
				iq_Cyl.Q.xSVBCmd		:= FALSE;
			END_IF
		END_IF

		IF iq_Cyl.Q.xSVACmd THEN
			IF xManCmd THEN
				iq_Cyl.Q.xSVACmd		:= FALSE;
				iq_Cyl.Q.xRetracted		:= FALSE;
				iq_Cyl.Q.xExtended		:= FALSE;
				iq_Timer.IN					:= TRUE;
			END_IF
		ELSE
			IF xManCmd THEN
				iq_Cyl.Q.xSVACmd		:= TRUE;
				iq_Cyl.Q.xSVBCmd		:= FALSE;
				iq_Cyl.Q.xRetracted		:= FALSE;
				iq_Cyl.Q.xExtended		:= FALSE;
				IF iq_Cyl.I.xValveOffRetract THEN
					iq_Cyl.Q.tTimeToExtend	:= T#0ms;
	 			ELSE
					iq_Cyl.Q.tTimeToRetract	:= T#0ms;
	 			END_IF
				iq_Timer.IN					:= TRUE;
			END_IF
		END_IF

		IF iq_Cyl.Q.xSVBCmd THEN
			IF xManCmdB THEN
				iq_Cyl.Q.xSVBCmd		:= FALSE;
				iq_Cyl.Q.xRetracted		:= FALSE;
				iq_Cyl.Q.xExtended		:= FALSE;
				iq_Timer.IN					:= TRUE;
			END_IF
		ELSE
			IF xManCmdB THEN
				iq_Cyl.Q.xSVBCmd		:= TRUE;
				iq_Cyl.Q.xSVACmd		:= FALSE;
				iq_Cyl.Q.xRetracted		:= FALSE;
				iq_Cyl.Q.xExtended		:= FALSE;
				IF iq_Cyl.I.xValveOffRetract THEN
					iq_Cyl.Q.tTimeToRetract	:= T#0ms;
	 			ELSE
					iq_Cyl.Q.tTimeToExtend	:= T#0ms;
	 			END_IF
				iq_Timer.IN					:= TRUE;
			END_IF
		END_IF
	END_IF

END_IF

END_FUNCTION

(* ---- FC_CylQ_2xSV_wBrake3.st ---- *)
(********************************************************************
 * COPYRIGHT -- Pro Pack Systems, Inc.
 ********************************************************************
 * Library: PPS_Cyl
 * File: FC_CylQ_1xSV_Basic.st
 * Author: PaulZ
 * Created: April 19, 2012
 ********************************************************************
 * Implementation of library PPS_Cyl
 ********************************************************************)

(* Controls the outputs for a Double SV Cylinder, with Brake *)
FUNCTION FC_CylQ_2xSV_wBrake3

IF iq_Cyl.I.diType = EN_Cyl_2xSV_Basic_WBrake OR
	iq_Cyl.I.diType = EN_Cyl_2xSV_Sensored_WBrake THEN

	IF NOT iq_Cyl.I.xEnManCntrl THEN (* When not in Manual Mode, control output *)

		IF iq_Cyl.IQ.xBrakeEn THEN
  			iq_Cyl.Q.xSVACmd		:= FALSE;
   			iq_Cyl.Q.xSVBCmd		:= FALSE;
   			iq_Cyl.Q.xSVBrakeCmd	:= TRUE;
			iq_Timer.IN					:= FALSE;
			iq_Cyl.IQ.xBrakeEn		:= FALSE;
   		END_IF

		IF iq_Cyl.IQ.xBrakeDis THEN
  			iq_Cyl.Q.xSVBrakeCmd	:= FALSE;
   			iq_Cyl.IQ.xBrakeDis		:= FALSE;
   		END_IF

		IF iq_Cyl.Q.xSVBrakeCmd THEN
  			iq_Cyl.IQ.xExtCmd		:= FALSE;
   			iq_Cyl.IQ.xRetCmd		:= FALSE;
   		END_IF

		IF iq_Cyl.I.xValveOffRetract THEN
			IF iq_Cyl.IQ.xExtCmd THEN
				iq_Cyl.Q.xSVACmd		:= TRUE;
				iq_Cyl.Q.xSVBCmd		:= FALSE;
				iq_Cyl.Q.xRetracted		:= FALSE;
				iq_Cyl.Q.xExtended		:= FALSE;
				iq_Cyl.Q.tTimeToExtend	:= T#0ms;
				iq_Timer.IN					:= TRUE;
				IF iq_Cyl.Q.xSVACmd AND NOT iq_Cyl.Q.xSVBCmd THEN
					iq_Cyl.IQ.xExtCmd		:= FALSE;
				END_IF
			END_IF

			IF iq_Cyl.IQ.xRetCmd THEN
				iq_Cyl.Q.xSVACmd		:= FALSE;
				iq_Cyl.Q.xSVBCmd		:= TRUE;
				iq_Cyl.Q.xExtended		:= FALSE;
				iq_Cyl.Q.xRetracted		:= FALSE;
				iq_Cyl.Q.tTimeToRetract	:= T#0ms;
				iq_Timer.IN					:= TRUE;
				IF NOT iq_Cyl.Q.xSVACmd AND iq_Cyl.Q.xSVBCmd THEN
					iq_Cyl.IQ.xRetCmd		:= FALSE;
				END_IF
			END_IF
		ELSE
			IF iq_Cyl.IQ.xExtCmd THEN
				iq_Cyl.Q.xSVACmd		:= FALSE;
				iq_Cyl.Q.xSVBCmd		:= TRUE;
				iq_Cyl.Q.xExtended		:= FALSE;
				iq_Cyl.Q.xRetracted		:= FALSE;
				iq_Cyl.Q.tTimeToExtend	:= T#0ms;
				iq_Timer.IN					:= TRUE;
				IF NOT iq_Cyl.Q.xSVACmd AND iq_Cyl.Q.xSVBCmd THEN
					iq_Cyl.IQ.xExtCmd		:= FALSE;
				END_IF
			END_IF

			IF iq_Cyl.IQ.xRetCmd THEN
				iq_Cyl.Q.xSVACmd		:= TRUE;
				iq_Cyl.Q.xSVBCmd		:= FALSE;
				iq_Cyl.Q.xExtended		:= FALSE;
				iq_Cyl.Q.xRetracted		:= FALSE;
				iq_Cyl.Q.tTimeToRetract	:= T#0ms;
				iq_Timer.IN					:= TRUE;
				IF iq_Cyl.Q.xSVACmd AND NOT iq_Cyl.Q.xSVBCmd THEN
					iq_Cyl.IQ.xRetCmd		:= FALSE;
				END_IF
			END_IF
		END_IF

	ELSE (* When in Manual Mode, control output *)

		IF xManBrake THEN
  			IF iq_Cyl.Q.xSVBrakeCmd THEN
   				iq_Cyl.Q.xSVBrakeCmd	:= FALSE;
			ELSE
			  	iq_Cyl.Q.xSVBrakeCmd	:= TRUE;
				iq_Cyl.Q.xSVACmd		:= FALSE;
				iq_Cyl.Q.xSVBCmd		:= FALSE;
			END_IF
		END_IF

		IF iq_Cyl.Q.xSVACmd THEN
			IF xManCmd THEN
				iq_Cyl.Q.xSVACmd		:= FALSE;
				iq_Cyl.Q.xRetracted		:= FALSE;
				iq_Cyl.Q.xExtended		:= FALSE;
				iq_Timer.IN					:= TRUE;
			END_IF
		ELSE
			IF xManCmd THEN
				iq_Cyl.Q.xSVACmd		:= TRUE;
				iq_Cyl.Q.xSVBCmd		:= FALSE;
				iq_Cyl.Q.xRetracted		:= FALSE;
				iq_Cyl.Q.xExtended		:= FALSE;
				IF iq_Cyl.I.xValveOffRetract THEN
					iq_Cyl.Q.tTimeToExtend	:= T#0ms;
	 			ELSE
					iq_Cyl.Q.tTimeToRetract	:= T#0ms;
	 			END_IF
				iq_Timer.IN					:= TRUE;
			END_IF
		END_IF

		IF iq_Cyl.Q.xSVBCmd THEN
			IF xManCmdB THEN
				iq_Cyl.Q.xSVBCmd		:= FALSE;
				iq_Cyl.Q.xRetracted		:= FALSE;
				iq_Cyl.Q.xExtended		:= FALSE;
				iq_Timer.IN					:= TRUE;
			END_IF
		ELSE
			IF xManCmdB THEN
				iq_Cyl.Q.xSVBCmd		:= TRUE;
				iq_Cyl.Q.xSVACmd		:= FALSE;
				iq_Cyl.Q.xRetracted		:= FALSE;
				iq_Cyl.Q.xExtended		:= FALSE;
				IF iq_Cyl.I.xValveOffRetract THEN
					iq_Cyl.Q.tTimeToRetract	:= T#0ms;
	 			ELSE
					iq_Cyl.Q.tTimeToExtend	:= T#0ms;
	 			END_IF
				iq_Timer.IN					:= TRUE;
			END_IF
		END_IF
	END_IF

END_IF

END_FUNCTION

(* ---- FB_CylCntrl2.st ---- *)
(********************************************************************
 * COPYRIGHT -- Pro Pack Systems, Inc.
 ********************************************************************
 * Library: PPS_Cyl
 * File: FB_CylCntrl2.st
 * Author: Paul Zurlinden
 * Created: April 16, 2012
 ********************************************************************
 * Implementation of library PPS_Cyl
 ********************************************************************)

(* Controls a pneumatic cylinder of the following types:
		EN_Cyl_1xSV_Basic
		EN_Cyl_1xSV_Sensored
		EN_Cyl_2xSV_Basic_NoBrake
		EN_Cyl_2xSV_Basic_WBrake
		EN_Cyl_2xSV_Sensored_NoBrake
		EN_Cyl_2xSV_Sensored_WBrake *)

FUNCTION_BLOCK FB_CylCntrl2

xMonitor :=	iq_CylCntrlInterface.I.diType = EN_Cyl_1xSV_Sensored OR
					iq_CylCntrlInterface.I.diType = EN_Cyl_2xSV_Sensored_NoBrake OR
					iq_CylCntrlInterface.I.diType = EN_Cyl_2xSV_Sensored_WBrake;

x2xSV	:= iq_CylCntrlInterface.I.diType = EN_Cyl_2xSV_Basic_NoBrake OR
				iq_CylCntrlInterface.I.diType = EN_Cyl_2xSV_Basic_WBrake OR
				iq_CylCntrlInterface.I.diType = EN_Cyl_2xSV_Sensored_NoBrake OR
				iq_CylCntrlInterface.I.diType = EN_Cyl_2xSV_Sensored_WBrake;

Timer(PT := iq_CylCntrlInterface.I.tTravelDel);

RT(CLK := iq_CylCntrlInterface.I.xManCmdA);
xManCmd	:= RT.Q;

RT_B(CLK := iq_CylCntrlInterface.I.xManCmdB);
xManCmdB := RT_B.Q;

RT_Brake(CLK := iq_CylCntrlInterface.I.xManBrake);
xManBrake := RT_Brake.Q;

RT_Air(CLK := iq_CylCntrlInterface.I.xAirOk);
FT_Air(CLK := iq_CylCntrlInterface.I.xAirOk);

(* Debounce Cylinder Position Sensors *)
IF xMonitor THEN
	aFB_SensExt[0](iq_DebounceInterface := iq_CylCntrlInterface.stSensorExt);
	aFB_SensExt[1](iq_DebounceInterface := iq_CylCntrlInterface.stSensorRet);

	RT_SensExt(CLK := iq_CylCntrlInterface.stSensorExt.I.xSignal);
	IF RT_SensExt.Q THEN
 		iq_CylCntrlInterface.Q.tTimeToExtend	:= Timer.ET;
	END_IF

	RT_SensRet(CLK := iq_CylCntrlInterface.stSensorRet.I.xSignal);
	IF RT_SensRet.Q THEN
 		iq_CylCntrlInterface.Q.tTimeToRetract	:= Timer.ET;
	END_IF
END_IF

xFaultSum	:= iq_CylCntrlInterface.Q.xFaultNoExt OR iq_CylCntrlInterface.Q.xFaultNoRet;

IF iq_CylCntrlInterface.I.xFaultReset THEN
	iq_CylCntrlInterface.Q.xFaultNoExt	:= FALSE;
	iq_CylCntrlInterface.Q.xFaultNoRet := FALSE;
END_IF

IF iq_CylCntrlInterface.I.xEnableFB THEN
	iq_CylCntrlInterface.Q.xFBActive	:= TRUE;

	(* Determine Cylinder Position when air is first turned on *)
	CASE iCheckAir OF
 		0:
			IF RT_Air.Q THEN
   				IF xMonitor OR x2xSV THEN
   					iCheckAir	:= 10;
				ELSE
					IF iq_CylCntrlInterface.I.xValveOffRetract THEN
   						IF iq_CylCntrlInterface.Q.xSVACmd THEN
							iq_CylCntrlInterface.Q.xExtended	:= TRUE;
							iq_CylCntrlInterface.Q.xRetracted	:= FALSE;
	 					ELSE
						   	iq_CylCntrlInterface.Q.xRetracted	:= TRUE;
							iq_CylCntrlInterface.Q.xExtended	:= FALSE;
	 					END_IF
					ELSE
						IF iq_CylCntrlInterface.Q.xSVACmd THEN
							iq_CylCntrlInterface.Q.xRetracted	:= TRUE;
							iq_CylCntrlInterface.Q.xExtended	:= FALSE;
	 					ELSE
						   	iq_CylCntrlInterface.Q.xExtended	:= TRUE;
							iq_CylCntrlInterface.Q.xRetracted	:= FALSE;
		 				END_IF
					END_IF
				END_IF
			END_IF

		10:
			IF xMonitor THEN
   				iCheckAir	:= 20;
			ELSE
				IF iq_CylCntrlInterface.I.xValveOffRetract THEN
   					IF iq_CylCntrlInterface.Q.xSVACmd THEN
						iq_CylCntrlInterface.Q.xExtended	:= TRUE;
						iq_CylCntrlInterface.Q.xRetracted	:= FALSE;
						iCheckAir										:= 0;
	 				ELSIF iq_CylCntrlInterface.Q.xSVBCmd THEN
					   	iq_CylCntrlInterface.Q.xRetracted	:= TRUE;
						iq_CylCntrlInterface.Q.xExtended	:= FALSE;
						iCheckAir										:= 0;
	 				END_IF
				ELSE
					IF iq_CylCntrlInterface.Q.xSVACmd THEN
						iq_CylCntrlInterface.Q.xRetracted	:= TRUE;
						iq_CylCntrlInterface.Q.xExtended	:= FALSE;
						iCheckAir										:= 0;
	 				ELSIF iq_CylCntrlInterface.Q.xSVBCmd THEN
					   	iq_CylCntrlInterface.Q.xExtended	:= TRUE;
						iq_CylCntrlInterface.Q.xRetracted	:= FALSE;
						iCheckAir										:= 0;
		 			END_IF
				END_IF
			END_IF

		20:
			IF iq_CylCntrlInterface.stSensorExt.Q.xCmd THEN
   				iq_CylCntrlInterface.Q.xExtended	:= TRUE;
				iq_CylCntrlInterface.Q.xRetracted	:= FALSE;
				iCheckAir										:= 0;
			END_IF

			IF iq_CylCntrlInterface.stSensorRet.Q.xCmd THEN
   				iq_CylCntrlInterface.Q.xRetracted	:= TRUE;
				iq_CylCntrlInterface.Q.xExtended	:= FALSE;
				iCheckAir										:= 0;
			END_IF

	END_CASE

	(* Fault Montiors *)
	FC_CylFM_1xSV_Basic(iq_CylCntrlInterface, Timer);
	FC_CylFM_1xSV_Sensored(iq_CylCntrlInterface, Timer);
	FC_CylFM_2xSV_Basic_NoBrake(iq_CylCntrlInterface, Timer);
	FC_CylFM_2xSV_Basic_wBrake(iq_CylCntrlInterface, Timer);
	FC_CylFM_2xSV_Sensored_NoBrake(iq_CylCntrlInterface, Timer);
	FC_CylFM_2xSV_Sensored_wBrake(iq_CylCntrlInterface, Timer);

	(* Control output *)
	IF iq_CylCntrlInterface.I.xEmergency OR xFaultSum OR FT_Air.Q THEN
		iq_CylCntrlInterface.Q.xSVACmd			:= FALSE;
		iq_CylCntrlInterface.Q.xSVBCmd			:= FALSE;
		iq_CylCntrlInterface.Q.xSVBrakeCmd	:= FALSE;
	ELSE
		FC_CylQ_1xSV(xManCmd, iq_CylCntrlInterface, Timer);
		FC_CylQ_2xSV_NoBrake(xManCmd, xManCmdB, iq_CylCntrlInterface, Timer);
		FC_CylQ_2xSV_wBrake(xManCmd, xManCmdB, xManBrake, iq_CylCntrlInterface, Timer);
	END_IF

	IF iq_CylCntrlInterface.I.xEmergency THEN
 		iq_CylCntrlInterface.Q.xExtended	:= FALSE;
  		iq_CylCntrlInterface.Q.xRetracted	:= FALSE;
  	END_IF

ELSE
	iq_CylCntrlInterface.Q.xFBActive			:= FALSE;
	iq_CylCntrlInterface.Q.xSVACmd			:= FALSE;
	iq_CylCntrlInterface.Q.xSVBCmd			:= FALSE;
 	iq_CylCntrlInterface.Q.xSVBrakeCmd	:= FALSE;
	iq_CylCntrlInterface.Q.xExtended		:= FALSE;
	iq_CylCntrlInterface.Q.xRetracted		:= FALSE;
	Timer.IN											:= FALSE;
END_IF

END_FUNCTION_BLOCK

(* ---- FB_CylCntrl3.st ---- *)
(********************************************************************
 * COPYRIGHT -- Pro Pack Systems, Inc.
 ********************************************************************
 * Library: PPS_Cyl
 * File: FB_CylCntrl3.st
 * Author: PaulZ
 * Created: March 14, 2013
 ********************************************************************
 * Implementation of library PPS_Cyl
 ********************************************************************)

(* Controls a pneumatic cylinder of the following types:
		EN_Cyl_1xSV_Basic
		EN_Cyl_1xSV_Sensored
		EN_Cyl_2xSV_Basic_NoBrake
		EN_Cyl_2xSV_Basic_WBrake
		EN_Cyl_2xSV_Sensored_NoBrake
		EN_Cyl_2xSV_Sensored_WBrake *)

FUNCTION_BLOCK FB_CylCntrl3

xMonitor :=	iq_CylCntrlInterface.I.diType = EN_Cyl_1xSV_Sensored OR
					iq_CylCntrlInterface.I.diType = EN_Cyl_2xSV_Sensored_NoBrake OR
					iq_CylCntrlInterface.I.diType = EN_Cyl_2xSV_Sensored_WBrake;

x2xSV	:= iq_CylCntrlInterface.I.diType = EN_Cyl_2xSV_Basic_NoBrake OR
				iq_CylCntrlInterface.I.diType = EN_Cyl_2xSV_Basic_WBrake OR
				iq_CylCntrlInterface.I.diType = EN_Cyl_2xSV_Sensored_NoBrake OR
				iq_CylCntrlInterface.I.diType = EN_Cyl_2xSV_Sensored_WBrake;

Timer(PT := iq_CylCntrlInterface.I.tTravelDel);

RT(CLK := iq_CylCntrlInterface.I.xManCmdA);
xManCmd	:= RT.Q;

RT_B(CLK := iq_CylCntrlInterface.I.xManCmdB);
xManCmdB := RT_B.Q;

RT_Brake(CLK := iq_CylCntrlInterface.I.xManBrake);
xManBrake := RT_Brake.Q;

RT_Air(CLK := iq_CylCntrlInterface.I.xAirOk);
FT_Air(CLK := iq_CylCntrlInterface.I.xAirOk);

(* Debounce Cylinder Position Sensors *)
IF xMonitor THEN
	aFB_SensExt[0](iq_DebounceInterface := iq_CylCntrlInterface.stSensorExt);
	aFB_SensExt[1](iq_DebounceInterface := iq_CylCntrlInterface.stSensorRet);

	RT_SensExt(CLK := iq_CylCntrlInterface.stSensorExt.I.xSignal);
	IF RT_SensExt.Q THEN
 		iq_CylCntrlInterface.Q.tTimeToExtend	:= Timer.ET;
	END_IF

	RT_SensRet(CLK := iq_CylCntrlInterface.stSensorRet.I.xSignal);
	IF RT_SensRet.Q THEN
 		iq_CylCntrlInterface.Q.tTimeToRetract	:= Timer.ET;
	END_IF
END_IF

xFaultSum	:= iq_CylCntrlInterface.Q.xFault;

IF iq_CylCntrlInterface.IQ.xFaultReset THEN
	iq_CylCntrlInterface.Q.xFault			:= FALSE;
	iq_CylCntrlInterface.Q.sFaultText		:= '';
	iq_CylCntrlInterface.IQ.xFaultReset		:= FALSE;
END_IF

IF iq_CylCntrlInterface.I.xEnableFB THEN
	iq_CylCntrlInterface.Q.xFBActive	:= TRUE;

	(* Determine Cylinder Position when air is first turned on *)
	CASE iCheckAir OF
 		0:
			IF RT_Air.Q THEN
   				IF xMonitor OR x2xSV THEN
   					iCheckAir	:= 10;
				ELSE
					IF iq_CylCntrlInterface.I.xValveOffRetract THEN
   						IF iq_CylCntrlInterface.Q.xSVACmd THEN
							iq_CylCntrlInterface.Q.xExtended	:= TRUE;
							iq_CylCntrlInterface.Q.xRetracted	:= FALSE;
	 					ELSE
						   	iq_CylCntrlInterface.Q.xRetracted	:= TRUE;
							iq_CylCntrlInterface.Q.xExtended	:= FALSE;
	 					END_IF
					ELSE
						IF iq_CylCntrlInterface.Q.xSVACmd THEN
							iq_CylCntrlInterface.Q.xRetracted	:= TRUE;
							iq_CylCntrlInterface.Q.xExtended	:= FALSE;
	 					ELSE
						   	iq_CylCntrlInterface.Q.xExtended	:= TRUE;
							iq_CylCntrlInterface.Q.xRetracted	:= FALSE;
		 				END_IF
					END_IF
				END_IF
			END_IF

		10:
			IF xMonitor THEN
   				iCheckAir	:= 20;
			ELSE
				IF iq_CylCntrlInterface.I.xValveOffRetract THEN
   					IF iq_CylCntrlInterface.Q.xSVACmd THEN
						iq_CylCntrlInterface.Q.xExtended	:= TRUE;
						iq_CylCntrlInterface.Q.xRetracted	:= FALSE;
						iCheckAir										:= 0;
	 				ELSIF iq_CylCntrlInterface.Q.xSVBCmd THEN
					   	iq_CylCntrlInterface.Q.xRetracted	:= TRUE;
						iq_CylCntrlInterface.Q.xExtended	:= FALSE;
						iCheckAir										:= 0;
	 				END_IF
				ELSE
					IF iq_CylCntrlInterface.Q.xSVACmd THEN
						iq_CylCntrlInterface.Q.xRetracted	:= TRUE;
						iq_CylCntrlInterface.Q.xExtended	:= FALSE;
						iCheckAir										:= 0;
	 				ELSIF iq_CylCntrlInterface.Q.xSVBCmd THEN
					   	iq_CylCntrlInterface.Q.xExtended	:= TRUE;
						iq_CylCntrlInterface.Q.xRetracted	:= FALSE;
						iCheckAir										:= 0;
		 			END_IF
				END_IF
			END_IF

		20:
			IF iq_CylCntrlInterface.stSensorExt.Q.xCmd THEN
   				iq_CylCntrlInterface.Q.xExtended	:= TRUE;
				iq_CylCntrlInterface.Q.xRetracted	:= FALSE;
				iCheckAir										:= 0;
			END_IF

			IF iq_CylCntrlInterface.stSensorRet.Q.xCmd THEN
   				iq_CylCntrlInterface.Q.xRetracted	:= TRUE;
				iq_CylCntrlInterface.Q.xExtended	:= FALSE;
				iCheckAir										:= 0;
			END_IF

	END_CASE

	(* Fault Montiors *)
	FC_CylFM_1xSV_Basic3(iq_CylCntrlInterface, Timer);
	FC_CylFM_1xSV_Sensored3(iq_CylCntrlInterface, Timer);
	FC_CylFM_2xSV_Basic_NoBrake3(iq_CylCntrlInterface, Timer);
	FC_CylFM_2xSV_Basic_wBrake3(iq_CylCntrlInterface, Timer);
	FC_CylFM_2xSV_Sensored_NoBrake3(iq_CylCntrlInterface, Timer);
	FC_CylFM_2xSV_Sensored_wBrake3(iq_CylCntrlInterface, Timer);

	(* Control output *)
	IF iq_CylCntrlInterface.I.xEmergency OR xFaultSum OR FT_Air.Q THEN
		iq_CylCntrlInterface.Q.xSVACmd			:= FALSE;
		iq_CylCntrlInterface.Q.xSVBCmd			:= FALSE;
		iq_CylCntrlInterface.Q.xSVBrakeCmd	:= FALSE;
	ELSE
		FC_CylQ_1xSV3(xManCmd, iq_CylCntrlInterface, Timer);
		FC_CylQ_2xSV_NoBrake3(xManCmd, xManCmdB, iq_CylCntrlInterface, Timer);
		FC_CylQ_2xSV_wBrake3(xManCmd, xManCmdB, xManBrake, iq_CylCntrlInterface, Timer);
	END_IF

	IF iq_CylCntrlInterface.I.xEmergency THEN
 		iq_CylCntrlInterface.Q.xExtended	:= FALSE;
  		iq_CylCntrlInterface.Q.xRetracted	:= FALSE;
  	END_IF

ELSE
	iq_CylCntrlInterface.Q.xFBActive			:= FALSE;
	iq_CylCntrlInterface.Q.xSVACmd			:= FALSE;
	iq_CylCntrlInterface.Q.xSVBCmd			:= FALSE;
 	iq_CylCntrlInterface.Q.xSVBrakeCmd	:= FALSE;
	iq_CylCntrlInterface.Q.xExtended		:= FALSE;
	iq_CylCntrlInterface.Q.xRetracted		:= FALSE;
	Timer.IN											:= FALSE;
END_IF

END_FUNCTION_BLOCK

(* ---- PPS_Cyl.fun ---- *)
(********************************************************************
 * COPYRIGHT -- Pro Pack Systems, Inc.
 ********************************************************************
 * Library: PPS_Cyl
 * File: PPS_Cyl.fun
 * Author: PaulZ
 * Created: April 16, 2012
 ********************************************************************
 * Functions and function blocks of library PPS_Cyl
 ********************************************************************)

FUNCTION_BLOCK FB_CylCntrl2 (*Controls a pneumatic cylinder with or without end of travel sensors*)
	VAR_IN_OUT
		iq_CylCntrlInterface : dtCylCntrlInterface2;
	END_VAR
	VAR
		RT : R_TRIG;
		RT_B : R_TRIG;
		xManCmdB : BOOL;
		RT_Brake : R_TRIG;
		xManBrake : BOOL;
		xManCmd : BOOL;
		Timer : TON;
		RT_Air : R_TRIG;
		FT_Air : F_TRIG;
		xFaultSum : BOOL;
		aFB_SensExt : ARRAY[0..1] OF FB_Debounce;
		RT_SensExt : R_TRIG;
		RT_SensRet : R_TRIG;
		xMonitor : BOOL;
		iCheckAir : INT;
		x2xSV : BOOL;
	END_VAR
END_FUNCTION_BLOCK

FUNCTION FC_CylFM_1xSV_Basic : BOOL (*Monitors Cylinder Fault for Single SV Cylinder*)
	VAR_IN_OUT
		iq_Cyl : dtCylCntrlInterface2;
		iq_Timer : TON;
	END_VAR
END_FUNCTION

FUNCTION FC_CylFM_1xSV_Basic3 : BOOL (*Monitors Cylinder Fault for Single SV Cylinder*)
	VAR_IN_OUT
		iq_Cyl : dtCylCntrlInterface3;
		iq_Timer : TON;
	END_VAR
END_FUNCTION

FUNCTION FC_CylFM_1xSV_Sensored : BOOL (*Monitors Cylinder Fault for Single SV Cylinder with Sensors*)
	VAR_IN_OUT
		iq_Cyl : dtCylCntrlInterface2;
		iq_Timer : TON;
	END_VAR
	VAR
		xFaultSum : BOOL;
	END_VAR
END_FUNCTION

FUNCTION FC_CylFM_1xSV_Sensored3 : BOOL (*Monitors Cylinder Fault for Single SV Cylinder with Sensors*)
	VAR_IN_OUT
		iq_Cyl : dtCylCntrlInterface3;
		iq_Timer : TON;
	END_VAR
	VAR
		xFaultSum : BOOL;
		sNoExtTxt : STRING[80] := ' did not extend';
		sNoRetTxt : STRING[80] := ' did not retract';
	END_VAR
END_FUNCTION

FUNCTION FC_CylFM_2xSV_Basic_NoBrake : BOOL (*Monitors Cylinder Fault for Double SV Cylinder*)
	VAR_IN_OUT
		iq_Cyl : dtCylCntrlInterface2;
		iq_Timer : TON;
	END_VAR
END_FUNCTION

FUNCTION FC_CylFM_2xSV_Basic_NoBrake3 : BOOL (*Monitors Cylinder Fault for Double SV Cylinder*)
	VAR_IN_OUT
		iq_Cyl : dtCylCntrlInterface3;
		iq_Timer : TON;
	END_VAR
END_FUNCTION

FUNCTION FC_CylFM_2xSV_Sensored_NoBrake : BOOL (*Monitors Cylinder Fault for Double SV Cylinder with Sensor and no Brake*)
	VAR_IN_OUT
		iq_Cyl : dtCylCntrlInterface2;
		iq_Timer : TON;
	END_VAR
	VAR
		xFaultSum : BOOL;
	END_VAR
END_FUNCTION

FUNCTION FC_CylFM_2xSV_Sensored_NoBrake3 : BOOL (*Monitors Cylinder Fault for Double SV Cylinder with Sensor and no Brake*)
	VAR_IN_OUT
		iq_Cyl : dtCylCntrlInterface3;
		iq_Timer : TON;
	END_VAR
	VAR
		xFaultSum : BOOL;
		sNoExtTxt : STRING[80] := ' did not extend';
		sNoRetTxt : STRING[80] := ' did not retract';
	END_VAR
END_FUNCTION

FUNCTION FC_CylFM_2xSV_Sensored_wBrake : BOOL (*Monitors Cylinder Fault for Double SV Cylinder with Sensors and Brake*)
	VAR_IN_OUT
		iq_Cyl : dtCylCntrlInterface2;
		iq_Timer : TON;
	END_VAR
	VAR
		xFaultSum : BOOL;
	END_VAR
END_FUNCTION

FUNCTION FC_CylFM_2xSV_Sensored_wBrake3 : BOOL (*Monitors Cylinder Fault for Double SV Cylinder with Sensors and Brake*)
	VAR_IN_OUT
		iq_Cyl : dtCylCntrlInterface3;
		iq_Timer : TON;
	END_VAR
	VAR
		xFaultSum : BOOL;
		sNoExtTxt : STRING[80] := ' did not extend';
		sNoRetTxt : STRING[80] := ' did not retract';
	END_VAR
END_FUNCTION

FUNCTION FC_CylQ_1xSV : BOOL (*Controls the outputs for a Single SV Cylinder*)
	VAR_INPUT
		xManCmd : BOOL;
	END_VAR
	VAR_IN_OUT
		iq_Cyl : dtCylCntrlInterface2;
		iq_Timer : TON;
	END_VAR
END_FUNCTION

FUNCTION FC_CylQ_1xSV3 : BOOL (*Controls the outputs for a Single SV Cylinder*)
	VAR_INPUT
		xManCmd : BOOL;
	END_VAR
	VAR_IN_OUT
		iq_Cyl : dtCylCntrlInterface3;
		iq_Timer : TON;
	END_VAR
END_FUNCTION

FUNCTION FC_CylQ_2xSV_NoBrake : BOOL (*Controls the outputs for a Doube SV Cylinder, no Brake*)
	VAR_INPUT
		xManCmd : BOOL;
		xManCmdB : BOOL;
	END_VAR
	VAR_IN_OUT
		iq_Cyl : dtCylCntrlInterface2;
		iq_Timer : TON;
	END_VAR
END_FUNCTION

FUNCTION FC_CylQ_2xSV_NoBrake3 : BOOL (*Controls the outputs for a Doube SV Cylinder, no Brake*)
	VAR_INPUT
		xManCmd : BOOL;
		xManCmdB : BOOL;
	END_VAR
	VAR_IN_OUT
		iq_Cyl : dtCylCntrlInterface3;
		iq_Timer : TON;
	END_VAR
END_FUNCTION

FUNCTION FC_CylQ_2xSV_wBrake : BOOL (*Controls the outputs for a Doube SV Cylinder, with Brake*)
	VAR_INPUT
		xManCmd : BOOL;
		xManCmdB : BOOL;
		xManBrake : BOOL;
	END_VAR
	VAR_IN_OUT
		iq_Cyl : dtCylCntrlInterface2;
		iq_Timer : TON;
	END_VAR
END_FUNCTION

FUNCTION FC_CylQ_2xSV_wBrake3 : BOOL (*Controls the outputs for a Doube SV Cylinder, with Brake*)
	VAR_INPUT
		xManCmd : BOOL;
		xManCmdB : BOOL;
		xManBrake : BOOL;
	END_VAR
	VAR_IN_OUT
		iq_Cyl : dtCylCntrlInterface3;
		iq_Timer : TON;
	END_VAR
END_FUNCTION

FUNCTION FC_CylFM_2xSV_Basic_wBrake : BOOL (*Monitors faults for a 2x SV, no Sensors, with Brake*)
	VAR_IN_OUT
		iq_Cyl : dtCylCntrlInterface2;
		iq_Timer : TON;
	END_VAR
END_FUNCTION

FUNCTION FC_CylFM_2xSV_Basic_wBrake3 : BOOL (*Monitors faults for a 2x SV, no Sensors, with Brake*)
	VAR_IN_OUT
		iq_Cyl : dtCylCntrlInterface3;
		iq_Timer : TON;
	END_VAR
END_FUNCTION

FUNCTION_BLOCK FB_CylCntrl3 (*Controls a pneumatic cylinder*)
	VAR_IN_OUT
		iq_CylCntrlInterface : dtCylCntrlInterface3;
	END_VAR
	VAR
		RT : R_TRIG;
		RT_B : R_TRIG;
		xManCmdB : BOOL;
		RT_Brake : R_TRIG;
		xManBrake : BOOL;
		xManCmd : BOOL;
		Timer : TON;
		RT_Air : R_TRIG;
		FT_Air : F_TRIG;
		xFaultSum : BOOL;
		aFB_SensExt : ARRAY[0..1] OF FB_Debounce;
		RT_SensExt : R_TRIG;
		RT_SensRet : R_TRIG;
		xMonitor : BOOL;
		iCheckAir : INT;
		x2xSV : BOOL;
	END_VAR
END_FUNCTION_BLOCK

(* ---- PPS_Cyl.var ---- *)
(********************************************************************
 * COPYRIGHT -- Pro Pack Systems, Inc.
 ********************************************************************
 * Library: PPS_Cyl
 * File: PPS_Cyl.var
 * Author: PaulZ
 * Created: April 16, 2012
 ********************************************************************
 * Constants of library PPS_Cyl
 ********************************************************************)

VAR CONSTANT

END_VAR
